FUNCTION_BLOCK Output
  (* Standard: 61499-2 *)
  (* Version 0.1, 2017-00-29, hpea485, UOA *)
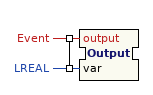
  EVENT_INPUT
    output WITH var;
  END_EVENT
  VAR_INPUT
    var : LREAL;
  END_VAR
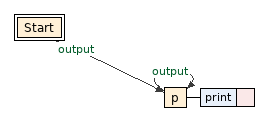
  EC_STATES
    Start;
    p : print;
  END_STATES
  EC_TRANSITIONS
    Start TO p := output;
    p TO p := output;
  END_TRANSITIONS
  ALGORITHM print IN C:
printf("New value: %f\n", me->var);
  END_ALGORITHM
END_FUNCTION_BLOCK
